(* IEC 61131-3 sources: sdplc/programs, 3 files *)

(* ---- control_flow.st ---- *)
(* all_control_flow.st — Every control flow construct
   Testing: IF, FOR, WHILE, REPEAT, CASE, EXIT, RETURN
   Compile: sdplc examples/all_control_flow.st
*)

FUNCTION Factorial : DINT
VAR_INPUT
    n : DINT;
END_VAR
VAR
    result : DINT := 1;
    i : DINT;
END_VAR

IF n <= 1 THEN
    Factorial := 1;
    RETURN;
END_IF;

FOR i := 2 TO n DO
    result := result * i;
END_FOR;

Factorial := result;

END_FUNCTION

PROGRAM ControlFlowDemo
VAR
    i : INT;
    j : INT;
    sum : DINT := 0;
    found : BOOL := FALSE;
    state : INT := 0;
    output : REAL := 0.0;
    limit : INT := 50;
END_VAR

(* ── FOR with BY step ── *)
FOR i := 0 TO 100 BY 5 DO
    sum := sum + i;
    IF sum > 500 THEN
        EXIT;
    END_IF;
END_FOR;

(* ── Nested FOR with EXIT ── *)
FOR i := 0 TO 9 DO
    FOR j := 0 TO 9 DO
        IF i * 10 + j >= limit THEN
            found := TRUE;
            EXIT;
        END_IF;
    END_FOR;
    IF found THEN
        EXIT;
    END_IF;
END_FOR;

(* ── WHILE ── *)
WHILE sum > 100 DO
    sum := sum / 2;
END_WHILE;

(* ── REPEAT / UNTIL ── *)
REPEAT
    sum := sum + 3;
UNTIL sum >= 50
END_REPEAT;

(* ── CASE with ranges and ELSE ── *)
CASE state OF
    0:
        output := 0.0;
    1..3:
        output := 25.0;
    4, 5:
        output := 50.0;
    6..9:
        output := 75.0;
ELSE
    output := 100.0;
END_CASE;

(* ── Deeply nested IF / ELSIF / ELSE ── *)
IF state = 0 THEN
    IF found THEN
        output := -1.0;
    ELSE
        output := -2.0;
    END_IF;
ELSIF state = 1 THEN
    output := 10.0;
ELSIF state = 2 THEN
    output := 20.0;
ELSE
    output := 99.0;
END_IF;

END_PROGRAM

(* ---- fb_library_demo.st ---- *)
(*
    Standard function block library demonstration.

    A small conveyor start/stop sequence that exercises every block in
    the SD-PLC standard library: the three timers, the three counters,
    both edge detectors and both latches. Run it with:

        cargo run --bin runtime -- programs/fb_library_demo.st --scan-time=50
*)
PROGRAM FbLibraryDemo
VAR
    (* Simulated field inputs, driven by the scan counter below so the
       program is self-exciting and needs no wiring to observe. *)
    scan_count : DINT := 0;
    start_button : BOOL := FALSE;
    stop_button : BOOL := FALSE;
    part_sensor : BOOL := FALSE;

    (* Function block instances — each one carries its own state. *)
    run_latch : RS;
    start_edge : R_TRIG;
    stop_edge : F_TRIG;
    warmup : TON;
    coast : TOF;
    horn : TP;
    parts : CTU;
    remaining : CTD;
    balance : CTUD;

    (* Outputs *)
    motor : BOOL := FALSE;
    conveyor_ready : BOOL := FALSE;
    brake : BOOL := FALSE;
    horn_on : BOOL := FALSE;
    warmup_elapsed : TIME;
    parts_done : BOOL := FALSE;
    parts_count : INT := 0;
    batch_empty : BOOL := FALSE;
    batch_reset : BOOL := FALSE;
END_VAR

scan_count := scan_count + 1;

(* Drive the simulated inputs: press start on scan 5, press and release
   stop around scan 200, and pulse the part sensor every 10 scans in
   between. Stop is released again so the horn's falling edge fires. *)
start_button := scan_count >= 5 AND scan_count < 10;
stop_button := scan_count >= 200 AND scan_count < 205;
part_sensor := (scan_count MOD 10) < 3 AND scan_count > 10 AND scan_count < 200;

(* Edge detection on the pushbuttons. *)
start_edge(CLK := start_button);
stop_edge(CLK := stop_button);

(* Reset-dominant latch: stop wins over start. *)
run_latch(S := start_edge.Q, R1 := stop_button);
motor := run_latch.Q1;

(* On-delay: the conveyor is only "ready" after the motor has run for
   two seconds continuously. *)
warmup(IN := motor, PT := T#2s);
conveyor_ready := warmup.Q;
warmup_elapsed := warmup.ET;

(* Off-delay: the brake stays engaged for 1.5s after the motor stops. *)
coast(IN := NOT motor, PT := T#1500ms);
brake := coast.Q;

(* Pulse: one 500ms horn blast on each falling edge of the stop button. *)
horn(IN := stop_edge.Q, PT := T#500ms);
horn_on := horn.Q;

(* Up counter: parts seen, Q latches once the batch of 12 is complete. *)
parts(CU := part_sensor, R := start_edge.Q, PV := 12);
parts_count := parts.CV;
parts_done := parts.Q;

(* Down counter: how many are left in the batch. *)
remaining(CD := part_sensor, LD := start_edge.Q, PV := 12);
batch_empty := remaining.Q;

(* Up/down counter: net balance of parts in against parts out. *)
balance(CU := part_sensor, CD := stop_button, R := start_edge.Q, PV := 12);
batch_reset := balance.QD;

END_PROGRAM

(* ---- flotation_tank.st ---- *)
PROGRAM FlotationTank
VAR
    cycle : DINT := 0;
    level : REAL := 50.0;
    air_flow : REAL := 30.0;
    feed_flow : REAL := 40.0;
    tailings_flow : REAL := 38.0;
    concentrate_grade : REAL := 82.0;
    target_level : REAL := 55.0;
    emergency_stop : BOOL := FALSE;
    motor_running : BOOL := TRUE;
    high_level : BOOL := FALSE;
    low_air : BOOL := FALSE;
END_VAR

cycle := cycle + 1;

high_level := level > 70.0;
low_air := air_flow < 20.0;

IF emergency_stop THEN
    motor_running := FALSE;
    air_flow := air_flow * 0.95;
ELSE
    motor_running := TRUE;
END_IF;

IF motor_running THEN
    IF level < target_level THEN
        tailings_flow := tailings_flow - 0.05;
    ELSE
        tailings_flow := tailings_flow + 0.05;
    END_IF;

    IF low_air THEN
        air_flow := air_flow + 0.25;
    ELSIF air_flow > 60.0 THEN
        air_flow := 60.0;
    ELSE
        air_flow := air_flow + 0.02;
    END_IF;
ELSE
    tailings_flow := tailings_flow * 0.98;
END_IF;

IF high_level THEN
    feed_flow := feed_flow - 0.10;
ELSE
    feed_flow := feed_flow + 0.02;
END_IF;

level := level + (feed_flow - tailings_flow) * 0.0005;
concentrate_grade := 82.0 + (air_flow - 25.0) * 0.03;

END_PROGRAM
